PROGRAM MAIN
VAR
	// flag to init robot
	g_robotInit :BOOL :=FALSE;
	
	// master robot
	g_masterRobot:FB_MasterRobot;
	
	// master robot information, export to other task or device
	m_masterStatus AT %Q* :ST_MasterStatus;
	
	// cart information, import from other task
	m_cartStatus AT %I*:ST_CartStatus;
	
	// slave robot information, import from other device
	m_slaveStatus AT %I*:ST_SlaveStatus;
	
END_VAR



IF g_robotInit =FALSE THEN
	g_masterRobot.Init();
	g_robotInit:=TRUE;
END_IF

g_masterRobot.run(m_cartStatus,m_slaveStatus);

END_PROGRAM

(* stored: Version 1.1.0.1, ProductVersion 3.1.4024.12
   POU MAIN: Id {6192c11b-cd6e-4883-b627-958acfb9caf3}, SpecialFunc None *)
